PROGRAM TemperatureControl
VAR
	fbTemperaturePIDControl	: FB_TemperaturePIDControl;
END_VAR

//fbTemperaturePIDControl();

END_PROGRAM

(* stored: Version 1.1.0.1, ProductVersion 3.1.4024.9
   POU TemperatureControl: Id {f71717d9-deae-438c-aba5-3161ba70bdae}, SpecialFunc None *)
